(* CoDeSys 2.3.9.41 project: Lab4b.pro *)
(* Libraries: Lab4.lib 12.11.15 19:02:24, STANDARD.LIB 5.6.98 12:03:02 *)

(* Task configuration *)
TASK Standard (PRIORITY := 0, INTERVAL := T#1ms);
	MAIN
END_TASK

(* Global variable list: Global_Variables *)
VAR_GLOBAL
END_VAR

VAR_GLOBAL CONSTANT
	F_TASK : INT := 1000;
	PERIOD_TASK : REAL := 0.001;
END_VAR

(* POU MAIN, ST *)
PROGRAM MAIN
VAR
END_VAR
SignalGenerator();
END_PROGRAM

(* POU SignalGenerator, FBD *)
PROGRAM SignalGenerator
VAR
	a : REAL := 0.5;
	offset : REAL := 0;
	w : REAL := 10;
	w2 : REAL := 10;
	w3 : REAL := 10;
	duty : REAL := 0.25;
	pwm : REAL := 0;
	Counter : t_count;
	I1 : Integrator;
	i_out : REAL;
	cnt : INT;
	sinus : REAL;
	sinus2 : REAL;
	sinus3 : REAL;
	LP1 : LowpassFilter;
	LP2 : LowpassFilter;
	LP3 : LowpassFilter;
	tau1 : INT := 10;
	tau2 : INT := 100;
	tau3 : INT := 1000;
	lp1_out : REAL;
	lp2_out : REAL;
	lp3_out : REAL;
	pt21 : SecondOrderLag;
	pt22 : SecondOrderLag;
	pt23 : SecondOrderLag;
	omega : REAL := 1;
	omega2 : REAL := 9.5916;
	omega3: REAL := 100;
	d : REAL := 0.2;
	pt21_out : REAL;
	pt22_out : REAL;
	pt23_out : REAL;
END_VAR
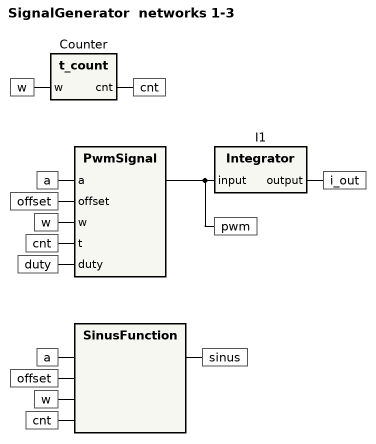
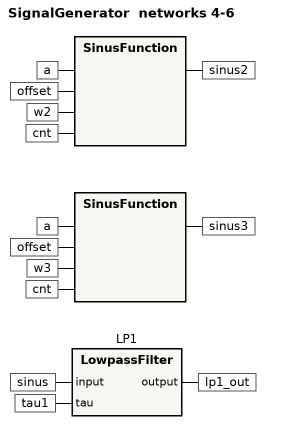
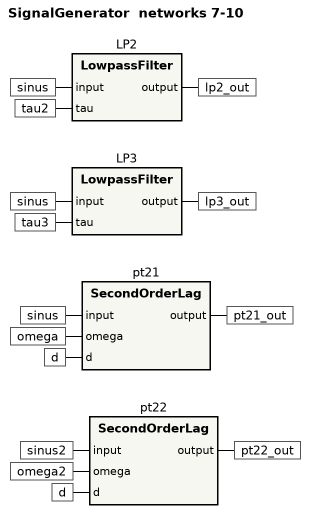
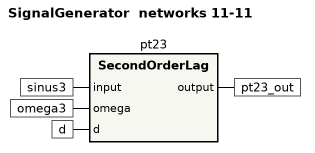
_FBD_ (* Function Block Diagram *)
NETWORK 1
	Counter:t_count(w: w) => cnt
NETWORK 2
	I1:Integrator(input: <PwmSignal(a: a, offset: offset, w: w, t: cnt, duty: duty) => pwm>) => i_out
NETWORK 3
	SinusFunction(a, offset, w, cnt) => sinus
NETWORK 4
	SinusFunction(a, offset, w2, cnt) => sinus2
NETWORK 5
	SinusFunction(a, offset, w3, cnt) => sinus3
NETWORK 6
	LP1:LowpassFilter(input: sinus, tau: tau1) => lp1_out
NETWORK 7
	LP2:LowpassFilter(input: sinus, tau: tau2) => lp2_out
NETWORK 8
	LP3:LowpassFilter(input: sinus, tau: tau3) => lp3_out
NETWORK 9
	pt21:SecondOrderLag(input: sinus, omega: omega, d: d) => pt21_out
NETWORK 10
	pt22:SecondOrderLag(input: sinus2, omega: omega2, d: d) => pt22_out
NETWORK 11
	pt23:SecondOrderLag(input: sinus3, omega: omega3, d: d) => pt23_out
_END_FBD_
(* the same logic as Structured Text *)
(* Network 1 *)
Counter(w := w);
cnt := Counter.cnt;
(* Network 2: see the listing above *)
(* Network 3 *)
sinus := SinusFunction(a, offset, w, cnt);
(* Network 4 *)
sinus2 := SinusFunction(a, offset, w2, cnt);
(* Network 5 *)
sinus3 := SinusFunction(a, offset, w3, cnt);
(* Network 6 *)
LP1(input := sinus, tau := tau1);
lp1_out := LP1.output;
(* Network 7 *)
LP2(input := sinus, tau := tau2);
lp2_out := LP2.output;
(* Network 8 *)
LP3(input := sinus, tau := tau3);
lp3_out := LP3.output;
(* Network 9 *)
pt21(input := sinus, omega := omega, d := d);
pt21_out := pt21.output;
(* Network 10 *)
pt22(input := sinus2, omega := omega2, d := d);
pt22_out := pt22.output;
(* Network 11 *)
pt23(input := sinus3, omega := omega3, d := d);
pt23_out := pt23.output;
END_PROGRAM

(* POU t_count, ST *)
FUNCTION_BLOCK t_count
VAR_INPUT
	w : REAL;
END_VAR
VAR_OUTPUT
	cnt : INT;
END_VAR
VAR
	t : INT := 0;
END_VAR
IF t < REAL_TO_INT(w*F_TASK) THEN
	t := t + 1;
ELSE
	t := 0;
END_IF
cnt := t;
END_FUNCTION_BLOCK
